// TIA Portal V20 export
// export: Created 2025-12-01T14:57:17.6847839Z, ExportSetting None, DisplayName Totally Integrated Automation Portal, DisplayVersion V20 Update 3, DisplayName TIA Portal Openness, DisplayVersion V20 Update 3, DisplayName TIA Portal Version Control Interface, DisplayVersion V20 Update 3, DisplayName STEP 7 Professional, DisplayVersion V20 Update 3, DisplayName STEP 7 Safety, DisplayVersion V20 Update 2, DisplayName WinCC Basic/Comfort/Advanced, DisplayVersion V20 Update 3, DisplayName WinCC Professional, DisplayVersion V20 Update 3, DisplayName WinCC Unified, DisplayVersion V20 Update 3
DATA_BLOCK "DB666_SIMUL"   // DB666
{ S7_Optimized_Access := 'FALSE' }
// stored: AutoNumber false
   VAR
      total_registros : Int := 100;
      offset_primero : Int := 8;
      offset_registros : Int := 2;
      siguiente_a_cargar : Int := 1;
      dato : Array[1..100] of Int;
   END_VAR
BEGIN
END_DATA_BLOCK
